FUNCTION_BLOCK FB_CTRL_OUT (* Basic Function Block Type *)
  (* Standard: 61499-2; Classification: Control Modules; Description: CTRL_OUT adds to the CI input the value of OFFSET and returns the result to Y if MANUAL = FALSE. If MANUAL is TRUE at output Y the input value of MAN_IN + OFFSET is issued. Y is always limited to the boundaries defined by LIM_L and LIM_H. If Y reaches one of the limits, then the output LIM is TRUE. CTRL_OUT can be used to build own rule modules. *)
  (* Version 0.0, 2011-08-23, 4DIAC-IDE, 4DIAC-Consortium *)
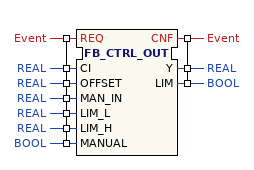
  EVENT_INPUT
    REQ WITH CI, OFFSET, MAN_IN, LIM_L, LIM_H, MANUAL; (* Normal Execution Request *)
  END_EVENT
  EVENT_OUTPUT
    CNF WITH LIM, Y; (* Execution Confirmation *)
  END_EVENT
  VAR_INPUT
    CI : REAL; (* input from controller *)
    OFFSET : REAL; (* output offset *)
    MAN_IN : REAL; (* manual input *)
    LIM_L : REAL; (* lower output limit *)
    LIM_H : REAL; (* upper output limit *)
    MANUAL : BOOL; (* switch for manual operation (TODO this could be also an event) *)
  END_VAR
  VAR_OUTPUT
    Y : REAL; (* Output event qualifier *)
    LIM : BOOL;
  END_VAR
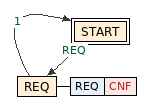
  EC_STATES
    START; (* Initial State *)
    REQ : REQ -> CNF; (* Normal execution *)
  END_STATES
  EC_TRANSITIONS
    START TO REQ := REQ;
    REQ TO START := 1;
  END_TRANSITIONS
  ALGORITHM REQ IN ST: (* Normally executed algorithm *)
Y := SEL(MANUAL, CI, MAN_IN) + OFFSET;

(* Limit the output *)
IF Y > LIM_L AND Y < LIM_H THEN
	LIM := FALSE;
ELSE
	Y := LIMIT(LIM_L, Y, LIM_H);
	LIM := TRUE;
END_IF;
  END_ALGORITHM
END_FUNCTION_BLOCK
